FUNCTION_BLOCK SKILL (* Composite Function Block Type *)
  (* Standard: 61499-2 *)
  (* Version 0.0, 1/31/2024, midxav, template *)
  PACKAGE Main;
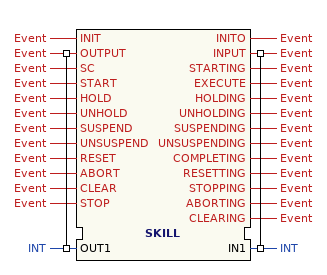
  EVENT_INPUT
    INIT;
    OUTPUT WITH OUT1;
    SC;
    START;
    HOLD;
    UNHOLD;
    SUSPEND;
    UNSUSPEND;
    RESET;
    ABORT;
    CLEAR;
    STOP;
  END_EVENT
  EVENT_OUTPUT
    INITO;
    INPUT WITH IN1;
    STARTING;
    EXECUTE;
    HOLDING;
    UNHOLDING;
    SUSPENDING;
    UNSUSPENDING;
    COMPLETING;
    RESETTING;
    STOPPING;
    ABORTING;
    CLEARING;
  END_EVENT
  VAR_INPUT
    OUT1 : INT;
  END_VAR
  VAR_OUTPUT
    IN1 : INT;
  END_VAR
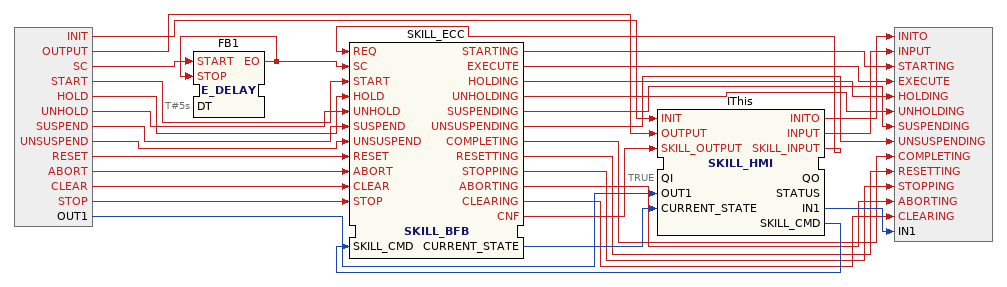
  FBS
    IThis : SKILL_HMI(QI := TRUE);
    SKILL_ECC : SKILL_BFB;
    FB1 : E_DELAY(DT := T#5s);
  END_FBS
  EVENT_CONNECTIONS
    SKILL_ECC.STARTING TO STARTING;
    SKILL_ECC.EXECUTE TO EXECUTE;
    SKILL_ECC.HOLDING TO HOLDING;
    SKILL_ECC.UNHOLDING TO UNHOLDING;
    SKILL_ECC.SUSPENDING TO SUSPENDING;
    SKILL_ECC.UNSUSPENDING TO UNSUSPENDING;
    SKILL_ECC.COMPLETING TO COMPLETING;
    SKILL_ECC.RESETTING TO RESETTING;
    SKILL_ECC.STOPPING TO STOPPING;
    SKILL_ECC.ABORTING TO ABORTING;
    SKILL_ECC.CLEARING TO CLEARING;
    INIT TO IThis.INIT;
    OUTPUT TO IThis.OUTPUT;
    SKILL_ECC.CNF TO IThis.SKILL_OUTPUT;
    IThis.INITO TO INITO;
    IThis.INPUT TO INPUT;
    IThis.SKILL_INPUT TO SKILL_ECC.REQ;
    SC TO FB1.START;
    FB1.EO TO FB1.STOP;
    FB1.EO TO SKILL_ECC.SC;
    START TO SKILL_ECC.START;
    HOLD TO SKILL_ECC.HOLD;
    UNHOLD TO SKILL_ECC.UNHOLD;
    SUSPEND TO SKILL_ECC.SUSPEND;
    UNSUSPEND TO SKILL_ECC.UNSUSPEND;
    RESET TO SKILL_ECC.RESET;
    ABORT TO SKILL_ECC.ABORT;
    CLEAR TO SKILL_ECC.CLEAR;
    STOP TO SKILL_ECC.STOP;
  END_CONNECTIONS
  DATA_CONNECTIONS
    OUT1 TO IThis.OUT1;
    SKILL_ECC.CURRENT_STATE TO IThis.CURRENT_STATE;
    IThis.IN1 TO IN1;
    IThis.SKILL_CMD TO SKILL_ECC.SKILL_CMD;
  END_CONNECTIONS
END_FUNCTION_BLOCK
